% RSLogix 500 project NASSCOM_BAK027.RSS, saved by version 8.30.00.16 %
PROJECT "UNTITLED"    % processor: Bul.1763 MicroLogix 1100 Series A %

PROGRAM FILES
  LAD 2   7 rungs

DATA FILES
  O0 OUTPUT  4 elements
  I1 INPUT  6 elements
  S2 STATUS  66 elements
  B3 BINARY  1 elements
  T4 TIMER  1 elements
  C5 COUNTER  1 elements
  R6 CONTROL  1 elements
  N7 INTEGER  10 elements
  F8 FLOAT  1 elements

LADDER 2
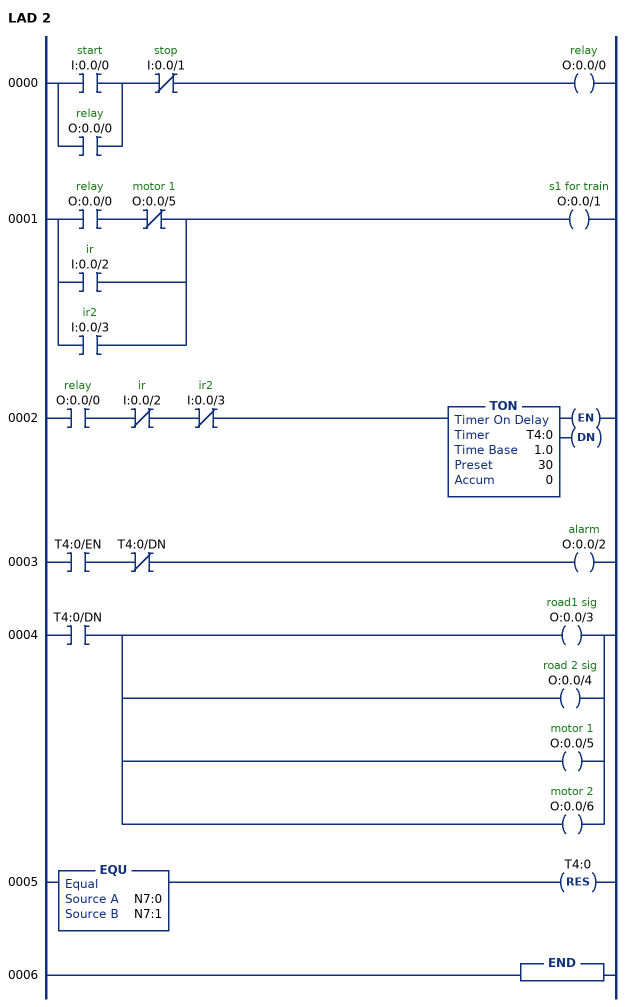
% Rung: 0 %
SOR BST XIC I:0.0/0 NXB XIC O:0.0/0 BND XIO I:0.0/1 OTE O:0.0/0 EOR
%   I:0.0/0  "start" %
%   O:0.0/0  "relay" %
%   I:0.0/1  "stop" %
% Rung: 1 %
SOR BST XIC O:0.0/0 XIO O:0.0/5 NXB BST XIC I:0.0/2 NXB XIC I:0.0/3 BND BND OTE O:0.0/1 EOR
%   O:0.0/0  "relay" %
%   O:0.0/5  "motor 1" %
%   I:0.0/2  "ir" %
%   I:0.0/3  "ir2" %
%   O:0.0/1  "s1 for train" %
% Rung: 2 %
SOR XIC O:0.0/0 XIO I:0.0/2 XIO I:0.0/3 TON T4:0 1.0 30 0 EOR
%   O:0.0/0  "relay" %
%   I:0.0/2  "ir" %
%   I:0.0/3  "ir2" %
% Rung: 3 %
SOR XIC T4:0/EN XIO T4:0/DN OTE O:0.0/2 EOR
%   O:0.0/2  "alarm" %
% Rung: 4 %
SOR XIC T4:0/DN BST OTE O:0.0/3 NXB BST OTE O:0.0/4 NXB BST OTE O:0.0/5 NXB OTE O:0.0/6 BND BND BND EOR
%   O:0.0/3  "road1 sig" %
%   O:0.0/4  "road 2 sig" %
%   O:0.0/5  "motor 1" %
%   O:0.0/6  "motor 2" %
% Rung: 5 %
SOR EQU N7:0 N7:1 RES T4:0 EOR
% Rung: 6 %
SOR END EOR

DATA TABLE (non-zero values as saved)
DATA T4
% .PRE .ACC %
% T4:0 % 30 0
DATA N7
% N7:0 % 2 0 0 0 0 0 0 0 0 0
